FUNCTION_BLOCK FB_JACK
VAR_INPUT
	bDefaultState: BOOL;
	bDepened_open1:BOOL:=TRUE;
	bDepened_open2:BOOL:=TRUE;
	bDepened_close1:BOOL:=TRUE;
	bDepened_close2:BOOL:=TRUE;
	sName:STRING;
	
	
END_VAR

VAR_OUTPUT
	JackStatus:E_JACK_STATUS:=E_JACK_STATUS.UNINIT ;
	
	bVALVE_OPEN: BOOL;
	bVALVE_CLOSE: BOOL;
	bError_Condition_open:BOOL;
	bError_Condition_close:BOOL;
	bERROR:BOOL:=FALSE;
END_VAR

VAR_IN_OUT
	
END_VAR
	
VAR
	bCMD_OPEN: BOOL;
	bMANUAL: BOOL;
	bCMD_OPEN_SWR: BOOL;
	bCMD_CLOSE_SWR: BOOL;
	bInit: BOOL:=FALSE;
	bOperationDone:BOOL:=FALSE;
	timerOpening:ton;
	timerClosing:ton;
	timeoutOpening:ton;
	timeoutClosing:ton;
	bSTARTUP: BOOL:=FALSE;
	rtrigMANUAL: R_TRIG;
	rtrig_OPEN_ERROR: R_TRIG;
	rtrig_CLOSE_ERROR: R_TRIG;
	rtrig_OPEN_CONDITION: R_TRIG;
	rtrig_CLOSE_CONDITION: R_TRIG;
	
	bSEN_OPEN: BOOL;
	bSEN_CLOSE: BOOL;
	bStepDone: BOOL;
END_VAR

IF NOT bSTARTUP THEN
	bCMD_OPEN:=bDefaultState;
	bSTARTUP:=TRUE;
END_IF

CASE JackStatus OF
	E_JACK_STATUS.UNINIT:
	IF bInit THEN
		JackStatus:=E_JACK_STATUS.INIT;
	END_IF
  
	E_JACK_STATUS.INIT:
	bInit:=FALSE;
	SFCReset:=TRUE;
	IF bCMD_OPEN THEN
		SFCReset:=FALSE;
		JackStatus:=E_JACK_STATUS.OPENING;
	ELSE
		SFCReset:=FALSE;
		JackStatus:=E_JACK_STATUS.CLOSING;
	END_IF
	
	E_JACK_STATUS.OPENING:
		open_jack();
		
	E_JACK_STATUS.CLOSING:
		close_jack();
	
	E_JACK_STATUS.OPENED:	
	IF NOT bCMD_OPEN THEN
		JackStatus:=E_JACK_STATUS.CLOSING;
	END_IF
	
	E_JACK_STATUS.CLOSED:	
	IF bCMD_OPEN THEN
		JackStatus:=E_JACK_STATUS.OPENING;
	END_IF
	
	E_JACK_STATUS.ERROR:
	IF bInit THEN
		JackStatus:=E_JACK_STATUS.INIT;
	END_IF
	//ee
			
END_CASE

ACTION _aCHECK_active:

IF bDepened_close1 AND bDepened_close2 THEN
	bStepDone:=TRUE;
ELSE
	JackStatus:=E_JACK_STATUS.ERROR;
	bERROR:=TRUE;
END_IF
END_ACTION

ACTION _aCHECK_active_1:
IF bDepened_open1 AND bDepened_open2 THEN
	bStepDone:=TRUE;
ELSE
	JackStatus:=E_JACK_STATUS.ERROR;
	bERROR:=TRUE;
END_IF
END_ACTION

ACTION _aCHECK_entry:
bStepDone:=FALSE;
bERROR:=FALSE;
END_ACTION

ACTION _aCHECK_entry_1:
bStepDone:=FALSE;
bERROR:=FALSE;
END_ACTION

ACTION _aCLOSE_active:

IF bSEN_CLOSE
OR CLOSE.t>T#5S
THEN
	bStepDone:=TRUE;
END_IF
END_ACTION

ACTION _aCLOSE_entry:
bStepDone:=FALSE;
bVALVE_OPEN:=FALSE;
END_ACTION

ACTION _aCLOSE_exit:
IF bSEN_CLOSE THEN
	JackStatus:=E_JACK_STATUS.CLOSED;
ELSE
	JackStatus:=E_JACK_STATUS.ERROR;
	bERROR:=TRUE;
END_IF
END_ACTION

ACTION _aOPEN_active:
IF bSEN_OPEN
OR OPEN.t>T#5S
THEN
	bStepDone:=TRUE;
END_IF
END_ACTION

ACTION _aOPEN_entry:
bStepDone:=FALSE;
bVALVE_OPEN:=TRUE;
END_ACTION

ACTION _aOPEN_exit:
IF bSEN_OPEN THEN
	JackStatus:=E_JACK_STATUS.OPENED;
ELSE
	JackStatus:=E_JACK_STATUS.ERROR;
	bERROR:=TRUE;
END_IF
END_ACTION

ACTION close_jack:
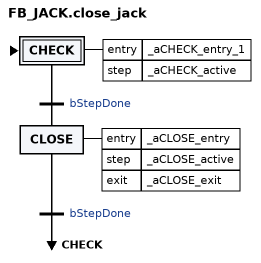
INITIAL_STEP CHECK:  // min time T#1s
    _aCHECK_entry_1(P1);  // entry action
    _aCHECK_active(N);  // step action
END_STEP
TRANSITION FROM CHECK TO CLOSE
    := bStepDone;
END_TRANSITION
STEP CLOSE:  // min time T#5s
    _aCLOSE_entry(P1);  // entry action
    _aCLOSE_active(N);  // step action
    _aCLOSE_exit(P0);  // exit action
END_STEP
TRANSITION FROM CLOSE TO CHECK
    := bStepDone;
END_TRANSITION
END_ACTION

ACTION open_jack:
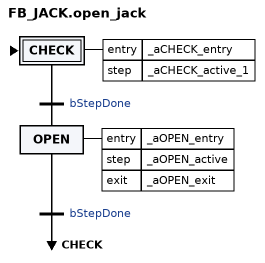
INITIAL_STEP CHECK:  // min time T#1s
    _aCHECK_entry(P1);  // entry action
    _aCHECK_active_1(N);  // step action
END_STEP
TRANSITION FROM CHECK TO OPEN
    := bStepDone;
END_TRANSITION
STEP OPEN:
    _aOPEN_entry(P1);  // entry action
    _aOPEN_active(N);  // step action
    _aOPEN_exit(P0);  // exit action
END_STEP
TRANSITION FROM OPEN TO CHECK
    := bStepDone;
END_TRANSITION
END_ACTION

END_FUNCTION_BLOCK

(* stored: Version 1.1.0.1, ProductVersion 3.1.4024.12
   POU FB_JACK: Id {facb1acf-b466-4a31-9974-a0d9880988b1}, SpecialFunc None
   Action _aCHECK_active: Id {265b8bd4-4fc5-4b20-8094-4371b72673b7}
   Action _aCHECK_active_1: Id {ca04d150-be0d-421e-a2c9-ea887380ed9f}
   Action _aCHECK_entry: Id {effb00a0-9146-4590-8416-08c1a91b2879}
   Action _aCHECK_entry_1: Id {dae13fde-49f1-482c-952e-175811d4a37b}
   Action _aCLOSE_active: Id {1529a8dd-50a5-4429-90db-11169e2033bb}
   Action _aCLOSE_entry: Id {427d9038-f34b-415f-a652-6d35fb096d6e}
   Action _aCLOSE_exit: Id {16010315-db04-4604-9f3e-4808b2f98608}
   Action _aOPEN_active: Id {e964eb8a-7e3a-4b49-bc11-574d6d0493e9}
   Action _aOPEN_entry: Id {0df89cc4-6f99-4662-81c7-8db72c8f59ae}
   Action _aOPEN_exit: Id {c4cd34a2-ec9f-44c6-a113-15e553b51a70}
   Action close_jack: Id {c3a58efc-c997-4828-a552-05fde68c3de9}
   Action open_jack: Id {12b33ed6-67a0-49c2-9392-61cd150320ae} *)
